(* CoDeSys 2.3 export: E_GABINET.EXP *)

(* POU Rooms/E_gabinet, ST *)
FUNCTION_BLOCK E_gabinet
VAR
	mainLamp:OnOff;
	Shader: ButtonTriggeredShader;
END_VAR
mainLamp(input:=E5_1b, output => E6_1);

shader(input:=E5_1a, shader:=shader_gabinet, openOut=>E2_1a, closeOut=>E2_1b);
END_FUNCTION_BLOCK
